// TIA Portal V19 export
TYPE "LAF_typeAxisParameters"
// stored: Access Published
   STRUCT
      manual : "LAF_typeAxisMannualParameters";
      production : "LAF_typeAxisProductionParameters";
      maintenance { S7_SetPoint := 'True'} : "LAF_typeAxisMaintanceParameters";
   END_STRUCT;
END_TYPE
